// TIA Portal V19 export
TYPE "ValvesInfo_UDT"
   STRUCT
      Act : Struct   // Out Info of Valve Monitor FB
         Count : DInt;   // Number of Activations
         Duration : Int;   // Duration of last activation (Count of 100Ms)
         AvgDuration : Int;   // Avg Duration of last 10 Activations
      END_STRUCT;
      DeAct : Struct
         Count : DInt;   // Number of De-Activations
         Duration : Int;   // Duration of last deactivation (Count of 100Ms)
         AvgDuration : Int;   // Duration of last deactivation (Count of 100Ms)
      END_STRUCT;
      RESET : Bool;   // Reset above Info from SCADA
   END_STRUCT;
END_TYPE
